// TIA Portal V20 export
// export: Created 2025-12-01T14:56:12.3409241Z, ExportSetting None, DisplayName Totally Integrated Automation Portal, DisplayVersion V20 Update 3, DisplayName TIA Portal Openness, DisplayVersion V20 Update 3, DisplayName TIA Portal Version Control Interface, DisplayVersion V20 Update 3, DisplayName STEP 7 Professional, DisplayVersion V20 Update 3, DisplayName STEP 7 Safety, DisplayVersion V20 Update 2, DisplayName WinCC Basic/Comfort/Advanced, DisplayVersion V20 Update 3, DisplayName WinCC Professional, DisplayVersion V20 Update 3, DisplayName WinCC Unified, DisplayVersion V20 Update 3
TYPE "EstadoZona"
   STRUCT
      Error_CBx : Bool;
      Resetear_CBx : Bool;
      Bit_02 : Bool;
      Bit_03 : Bool;
      Bit_04 : Bool;
      Bit_05 : Bool;
      Bit_06 : Bool;
      Bit_07 : Bool;
      Marcha_CBx : Bool;
      PerReset_CBx : Bool;
      Manual_CBx : Bool;
      Automatico_CBx : Bool;
      Mantenimiento_CBx : Bool;   // Antiguo Remoto
      Rearme_CBx : Bool;
      Paro_CBx : Bool;
      ParoBlando_CBx : Bool;
   END_STRUCT;
END_TYPE
